FUNCTION_BLOCK StartAtMainTask EXTENDS TcoCore.TcoTask 
VAR
    {attribute 'hide'} 
	_progress : INT := 0;
    {attribute 'hide'} 
	_infoTimer :  TON;
    {attribute 'hide'} 
	_errorTimer :  TON;
    {attribute 'hide'} 
	_varInfo : __SYSTEM.VAR_INFO;
    {attribute 'hide'} 
	_sb : TcoCore.StringBuilder;
	{attribute 'hide'}
	_blink:TcoUtilities.TcoBlinker(THIS^);
END_VAR

VAR_IN_OUT
    inoConfig 	: TcoIrc5_Config_v_1_x_x;
	inoControl 	: TcoIrc5_Control_v_1_x_x;
	inoStatus 	: TcoIrc5_Status_v_1_x_x;	
END_VAR

IF Execute() THEN 
	_blink(inOnTime:=T#500MS,inOffTime:=T#500MS);

	IF _progress = 0 THEN
		IF NOT __ISVALIDREF(inoControl) THEN
			_varInfo :=__VARINFO(inoControl);
			Messenger.Programming(_sb.Clear().Append('<#Invalid reference: #>').Append(_varInfo.Symbol).ToString()).Pin();
		ELSIF NOT __ISVALIDREF(inoConfig) THEN                                                  
			_varInfo :=__VARINFO(inoConfig);                                                    
			Messenger.Programming(_sb.Clear().Append('<#Invalid reference: #>').Append(_varInfo.Symbol).ToString()).Pin();
		ELSIF NOT __ISVALIDREF(inoStatus) THEN                                                  
			_varInfo :=__VARINFO(inoStatus);                                                    
			Messenger.Programming(_sb.Clear().Append('<#Invalid reference: #>').Append(_varInfo.Symbol).ToString()).Pin();
		ELSE
			_progress := _progress + 1;
		END_IF

	END_IF
	IF _progress = 1 THEN
	
		
		inoControl.StartAtMain :=   _blink.outQ;
		
		IF inoStatus.State.PpMoved AND NOT inoStatus.State.SystemInputBusy THEN
			inoControl.StartAtMain :=FALSE;
			_progress:=0;
		END_IF
	END_IF
    DoneWhen(inoStatus.State.PpMoved AND NOT inoStatus.State.SystemInputBusy);
    CallTimers(TRUE);
	
	THIS^.ThrowWhen(_errorTimer.Q);
	
END_IF;

METHOD CallTimers
VAR_INPUT
	inValue : BOOL;
END_VAR
IF  __ISVALIDREF(inoConfig) THEN  
_infoTimer(IN := inValue, PT := THIS^.inoConfig.InfoTime);
_errorTimer(IN := inValue, PT := THIS^.inoConfig.ErrorTime);
END_IF;
END_METHOD

METHOD PUBLIC FB_init : BOOL
VAR_INPUT
    bInitRetains : BOOL; // if TRUE, the retain variables are initialized (warm start / cold start)
    bInCopyCode : BOOL; // if TRUE, the instance afterwards gets moved into the copy code (online change)
  	ParentObject : ITcoObject;	
END_VAR
END_METHOD

(*~
	<docu>
		<summary>
			Executes when task is aborted.
		</summary>			
	</docu>	
~*)
METHOD PROTECTED OnAbort
IF  __ISVALIDREF(inoStatus) THEN   THIS^.inoStatus.ActionDescription := '<#Start at Main was aborted, while not yet completed!#>';END_IF;
END_METHOD

(*~
	<docu>
		<summary>
			Executes when task reaches the ```Done``` state .
		</summary>			
	</docu>	
~*)
METHOD PROTECTED OnDone
IF  __ISVALIDREF(inoStatus) THEN  THIS^.inoStatus.ActionDescription := '<#Start at Main was completed successfully.#>';END_IF;
END_METHOD

(*~
	<docu>
		<summary>
			Executes when task reaches the ```Error``` state.
			<para>
				Do not confuse with <see cref="PlcDocu.TcoCore.TcoTask.WhileError()"/>, that is called cyclically until '''Error''' state is left.
			</para>
		</summary>			
	</docu>	
~*)
METHOD PROTECTED OnError
IF  __ISVALIDREF(inoStatus) THEN   THIS^.inoStatus.ActionDescription := '<#Start at Main finished with error.#>'; END_IF;
END_METHOD

METHOD PROTECTED OnStart
IF  __ISVALIDREF(inoStatus) THEN  THIS^.inoStatus.ActionDescription := '<#Start at Main started.#>'; END_IF;
END_METHOD

(*~
	<docu>
		<summary>
			Restores this instance to the Ready state. Can be called explicitly or from within one of the restore mechanisms.
			<para>
				See also <see cref="PlcDocu.TcoCore.TcoTask.AutoRestorable()"/>
			</para>
		</summary>			
	</docu>	
~*)
METHOD Restore : ITcoRestorable
SUPER^.Restore();
_progress := 0;
CallTimers(FALSE);
Messenger.UnPin();
END_METHOD

END_FUNCTION_BLOCK

(* stored: Version 1.1.0.1, ProductVersion 3.1.4024.12
   POU StartAtMainTask: Id {213bca30-5c03-0b43-34d1-c9e329dd4949}, SpecialFunc None
   Method CallTimers: Id {1719c2ef-baa0-044b-0467-4fd5ea8c4dbd}
   Method FB_init: Id {4091c726-117b-0a54-0c35-f340ad84a8d6}
   Method OnAbort: Id {648f203f-ea9c-0794-0d1e-933a958beb02}
   Method OnDone: Id {f331caa4-3ef4-09ab-25b6-a64d3499162b}
   Method OnError: Id {8a4572b6-c7d2-0503-06c2-d46ef44b96b1}
   Method OnStart: Id {60c4182e-dbf9-0425-1f82-e9b4d5d14b73}
   Method Restore: Id {a7a95e8a-0af2-00b6-33a7-43a2c838d10a} *)
